// SIMATIC S7-200 SMART project (STEP 7-Micro/WIN SMART), CPU SR60

SYMBOL_TABLE A_手动
手动_测试_故障蜂鸣器1     V100.0
手动_测试_故障蜂鸣器2     V100.1
手动_测试_故障蜂鸣器3     V100.2
手动_测试_故障蜂鸣器4     V100.3
手动_测试_故障蜂鸣器5     V100.4
手动_测试_运行指示灯1     V100.5
手动_测试_运行指示灯2     V100.6
手动_测试_运行指示灯3     V100.7
手动_测试_运行指示灯4     V101.0
手动_测试_运行指示灯5     V101.1
手动_测试_停机指示灯1     V101.2
手动_测试_停机指示灯2     V101.3
手动_测试_停机指示灯3     V101.4
手动_测试_停机指示灯4     V101.5
手动_测试_停机指示灯5     V101.6
手动_测试_清洗吹扫指示1    V101.7
手动_测试_清洗吹扫指示2    V102.0
手动_测试_清洗吹扫指示3    V102.1
手动_测试_清洗吹扫指示4    V102.2
手动_测试_清洗吹扫指示5    V102.3
手动_测试_螺杆启停1      V102.4
手动_测试_螺杆启停2      V102.5
手动_测试_螺杆启停3      V102.6
手动_测试_螺杆启停4      V102.7
手动_测试_螺杆启停5      V103.0
手动_测试_入口阀1       V103.1
手动_测试_入口阀2       V103.2
手动_测试_入口阀3       V103.3
手动_测试_入口阀4       V103.4
手动_测试_入口阀5       V103.5
手动_测试_清洗阀1       V103.6
手动_测试_清洗阀2       V103.7
手动_测试_清洗阀3       V104.0
手动_测试_清洗阀4       V104.1
手动_测试_清洗阀5       V104.2
手动_测试_吹扫阀1       V104.3
手动_测试_吹扫阀2       V104.4
手动_测试_吹扫阀3       V104.5
手动_测试_吹扫阀4       V104.6
手动_测试_吹扫阀5       V104.7
END_SYMBOL_TABLE

SYMBOL_TABLE 系统符号
Always_On        SM0.0    // 始终接通
END_SYMBOL_TABLE

SYMBOL_TABLE A_自动
启动标志位1           V120.0
启动标志位2           V120.1
启动标志位3           V120.2
启动标志位4           V120.3
启动标志位5           V120.4
停机标志位1           V120.5
停机标志位2           V120.6
停机标志位3           V120.7
停机标志位4           V121.0
停机标志位5           V121.1
复位标志位1           V121.2
复位标志位2           V121.3
复位标志位3           V121.4
复位标志位4           V121.5
复位标志位5           V121.6
急停标志位1           V121.7
急停标志位2           V122.0
急停标志位3           V122.1
急停标志位4           V122.2
急停标志位5           V122.3
故障标志位1           V122.4
故障标志位2           V122.5
故障标志位3           V122.6
故障标志位4           V122.7
故障标志位5           V123.0
异常标志位1           V123.1
异常标志位2           V123.2
异常标志位3           V123.3
异常标志位4           V123.4
异常标志位5           V123.5
步骤延时触发1          V123.6
步骤延时触发2          V123.7
步骤延时触发3          V124.0
步骤延时触发4          V124.1
步骤延时触发5          V124.2
步骤延时定时器1         T37
步骤延时定时器2         T38
步骤延时定时器3         T39
步骤延时定时器4         T40
步骤延时定时器5         T41
启动前吹扫定时器1        T42
启动前吹扫定时器2        T43
启动前吹扫定时器3        T44
启动前吹扫定时器4        T45
启动前吹扫定时器5        T46
停机清洗定时器1         T47
停机清洗定时器2         T48
停机清洗定时器3         T49
停机清洗定时器4         T50
停机清洗定时器5         T51
停机吹扫定时器1         T52
停机吹扫定时器2         T53
停机吹扫定时器3         T54
停机吹扫定时器4         T55
停机吹扫定时器5         T56
自动步骤1            VW250
自动步骤2            VW252
自动步骤3            VW254
自动步骤4            VW256
自动步骤5            VW258
启动前吹扫时间_变量1      VW260
启动前吹扫时间_变量2      VW262
启动前吹扫时间_变量3      VW264
启动前吹扫时间_变量4      VW266
启动前吹扫时间_变量5      VW268
启动前吹扫时间_变量6      VW270
启动前吹扫时间_变量7      VW272
启动前吹扫时间_变量8      VW274
启动前吹扫时间_变量9      VW276
启动前吹扫时间_变量10     VW278
停机清洗时间_变量1       VW280
停机清洗时间_变量2       VW282
停机清洗时间_变量3       VW284
停机清洗时间_变量4       VW286
停机清洗时间_变量5       VW288
停机清洗时间_变量6       VW290
停机清洗时间_变量7       VW292
停机清洗时间_变量8       VW294
停机清洗时间_变量9       VW296
停机清洗时间_变量10      VW298
停机吹扫时间_变量1       VW300
停机吹扫时间_变量2       VW302
停机吹扫时间_变量3       VW304
停机吹扫时间_变量4       VW306
停机吹扫时间_变量5       VW308
停机吹扫时间_变量6       VW310
停机吹扫时间_变量7       VW312
停机吹扫时间_变量8       VW314
停机吹扫时间_变量9       VW316
停机吹扫时间_变量10      VW318
END_SYMBOL_TABLE

SYMBOL_TABLE A_参数显示_VW
启动前吹扫时间_显示1      VW500
启动前吹扫时间_显示2      VW502
启动前吹扫时间_显示3      VW504
启动前吹扫时间_显示4      VW506
启动前吹扫时间_显示5      VW508
停机清洗时间_显示1       VW510
停机清洗时间_显示2       VW512
停机清洗时间_显示3       VW514
停机清洗时间_显示4       VW516
停机清洗时间_显示5       VW518
停机吹扫时间_显示1       VW520
停机吹扫时间_显示2       VW522
停机吹扫时间_显示3       VW524
停机吹扫时间_显示4       VW526
停机吹扫时间_显示5       VW528
END_SYMBOL_TABLE

SYMBOL_TABLE A_参数设置_VD
目标真空1            VD900
目标真空2            VD904
目标真空3            VD908
目标真空4            VD912
目标真空5            VD916
入口压变上限1          VD920
入口温变上限1          VD924
冷却温变上限1          VD928
磁翻板液位上限1         VD932
入口压变上限2          VD936
入口温变上限2          VD940
冷却温变上限2          VD944
磁翻板液位上限2         VD948
入口压变上限3          VD952
入口温变上限3          VD956
冷却温变上限3          VD960
磁翻板液位上限3         VD964
入口压变上限4          VD968
入口温变上限4          VD972
冷却温变上限4          VD976
磁翻板液位上限4         VD980
入口压变上限5          VD984
入口温变上限5          VD988
冷却温变上限5          VD992
磁翻板液位上限5         VD996
END_SYMBOL_TABLE

SYMBOL_TABLE A_参数设置_VW
启动前吹扫时间_设置1      VW400
启动前吹扫时间_设置2      VW402
启动前吹扫时间_设置3      VW404
启动前吹扫时间_设置4      VW406
启动前吹扫时间_设置5      VW408
停机清洗时间_设置1       VW410
停机清洗时间_设置2       VW412
停机清洗时间_设置3       VW414
停机清洗时间_设置4       VW416
停机清洗时间_设置5       VW418
停机吹扫时间_设定1       VW420
停机吹扫时间_设定2       VW422
停机吹扫时间_设定3       VW424
停机吹扫时间_设定4       VW426
停机吹扫时间_设定5       VW428
END_SYMBOL_TABLE

SYMBOL_TABLE A_参数显示_VD
入口压力值1           VD600
入口温度值1           VD604
冷却温度值1           VD608
磁翻板液位值1          VD612
入口压力值2           VD616
入口温度值2           VD620
冷却温度值2           VD624
磁翻板液位值2          VD628
入口压力值3           VD632
入口温度值3           VD636
冷却温度值3           VD640
磁翻板液位值3          VD644
入口压力值4           VD648
入口温度值4           VD652
冷却温度值4           VD656
磁翻板液位值4          VD660
入口压力值5           VD664
入口温度值5           VD668
冷却温度值5           VD672
磁翻板液位值5          VD676
END_SYMBOL_TABLE

SUBROUTINE_BLOCK A_手动:SBR1
TITLE=子程序注释
BEGIN
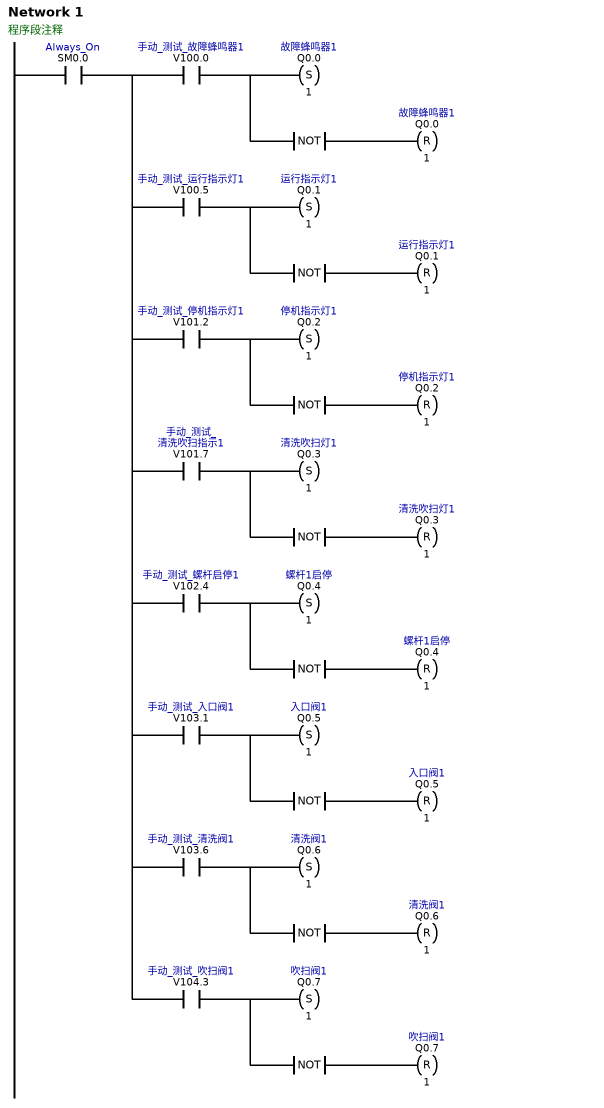
Network 1
// 程序段注释
LD     Always_On:SM0.0
LPS
A      手动_测试_故障蜂鸣器1:V100.0
S      故障蜂鸣器1:Q0.0, 1
NOT
R      故障蜂鸣器1:Q0.0, 1
LRD
A      手动_测试_运行指示灯1:V100.5
S      运行指示灯1:Q0.1, 1
NOT
R      运行指示灯1:Q0.1, 1
LRD
A      手动_测试_停机指示灯1:V101.2
S      停机指示灯1:Q0.2, 1
NOT
R      停机指示灯1:Q0.2, 1
LRD
A      手动_测试_清洗吹扫指示1:V101.7
S      清洗吹扫灯1:Q0.3, 1
NOT
R      清洗吹扫灯1:Q0.3, 1
LRD
A      手动_测试_螺杆启停1:V102.4
S      螺杆1启停:Q0.4, 1
NOT
R      螺杆1启停:Q0.4, 1
LRD
A      手动_测试_入口阀1:V103.1
S      入口阀1:Q0.5, 1
NOT
R      入口阀1:Q0.5, 1
LRD
A      手动_测试_清洗阀1:V103.6
S      清洗阀1:Q0.6, 1
NOT
R      清洗阀1:Q0.6, 1
LPP
A      手动_测试_吹扫阀1:V104.3
S      吹扫阀1:Q0.7, 1
NOT
R      吹扫阀1:Q0.7, 1
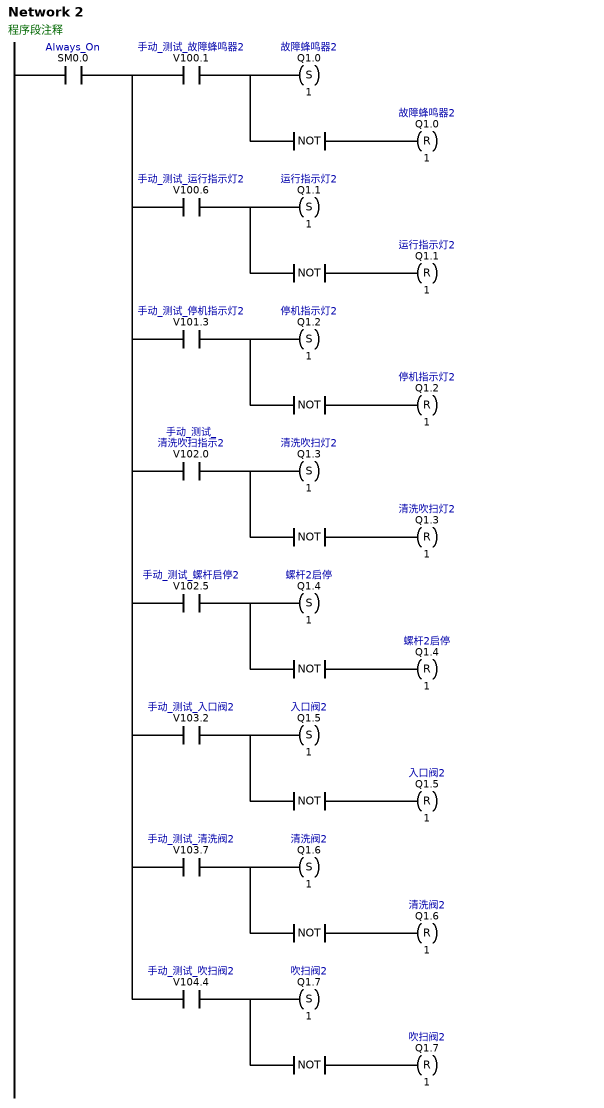
Network 2
// 程序段注释
LD     Always_On:SM0.0
LPS
A      手动_测试_故障蜂鸣器2:V100.1
S      故障蜂鸣器2:Q1.0, 1
NOT
R      故障蜂鸣器2:Q1.0, 1
LRD
A      手动_测试_运行指示灯2:V100.6
S      运行指示灯2:Q1.1, 1
NOT
R      运行指示灯2:Q1.1, 1
LRD
A      手动_测试_停机指示灯2:V101.3
S      停机指示灯2:Q1.2, 1
NOT
R      停机指示灯2:Q1.2, 1
LRD
A      手动_测试_清洗吹扫指示2:V102.0
S      清洗吹扫灯2:Q1.3, 1
NOT
R      清洗吹扫灯2:Q1.3, 1
LRD
A      手动_测试_螺杆启停2:V102.5
S      螺杆2启停:Q1.4, 1
NOT
R      螺杆2启停:Q1.4, 1
LRD
A      手动_测试_入口阀2:V103.2
S      入口阀2:Q1.5, 1
NOT
R      入口阀2:Q1.5, 1
LRD
A      手动_测试_清洗阀2:V103.7
S      清洗阀2:Q1.6, 1
NOT
R      清洗阀2:Q1.6, 1
LPP
A      手动_测试_吹扫阀2:V104.4
S      吹扫阀2:Q1.7, 1
NOT
R      吹扫阀2:Q1.7, 1
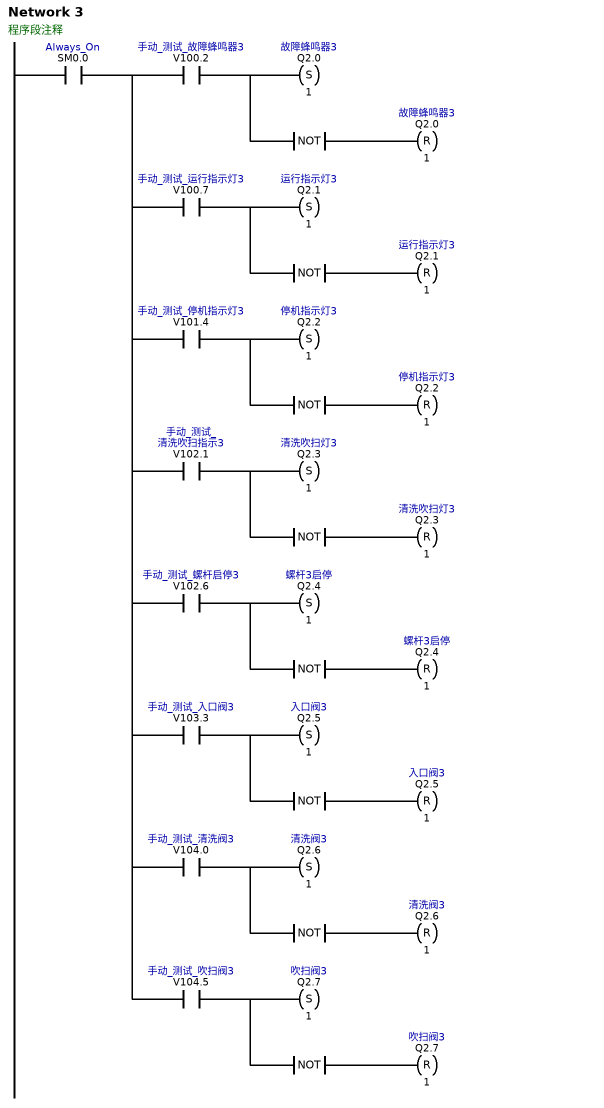
Network 3
// 程序段注释
LD     Always_On:SM0.0
LPS
A      手动_测试_故障蜂鸣器3:V100.2
S      故障蜂鸣器3:Q2.0, 1
NOT
R      故障蜂鸣器3:Q2.0, 1
LRD
A      手动_测试_运行指示灯3:V100.7
S      运行指示灯3:Q2.1, 1
NOT
R      运行指示灯3:Q2.1, 1
LRD
A      手动_测试_停机指示灯3:V101.4
S      停机指示灯3:Q2.2, 1
NOT
R      停机指示灯3:Q2.2, 1
LRD
A      手动_测试_清洗吹扫指示3:V102.1
S      清洗吹扫灯3:Q2.3, 1
NOT
R      清洗吹扫灯3:Q2.3, 1
LRD
A      手动_测试_螺杆启停3:V102.6
S      螺杆3启停:Q2.4, 1
NOT
R      螺杆3启停:Q2.4, 1
LRD
A      手动_测试_入口阀3:V103.3
S      入口阀3:Q2.5, 1
NOT
R      入口阀3:Q2.5, 1
LRD
A      手动_测试_清洗阀3:V104.0
S      清洗阀3:Q2.6, 1
NOT
R      清洗阀3:Q2.6, 1
LPP
A      手动_测试_吹扫阀3:V104.5
S      吹扫阀3:Q2.7, 1
NOT
R      吹扫阀3:Q2.7, 1
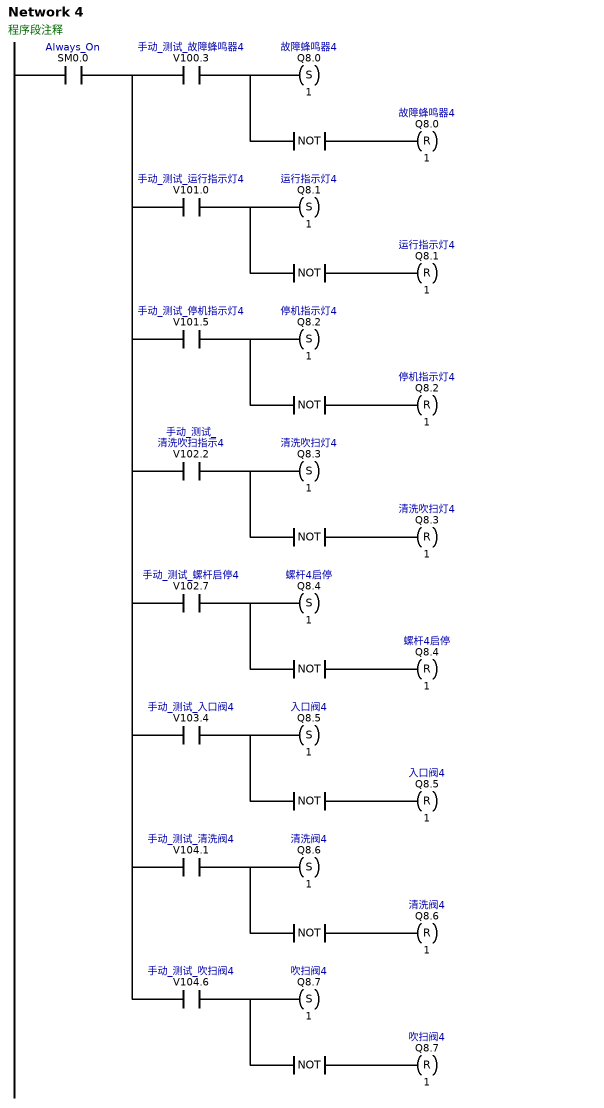
Network 4
// 程序段注释
LD     Always_On:SM0.0
LPS
A      手动_测试_故障蜂鸣器4:V100.3
S      故障蜂鸣器4:Q8.0, 1
NOT
R      故障蜂鸣器4:Q8.0, 1
LRD
A      手动_测试_运行指示灯4:V101.0
S      运行指示灯4:Q8.1, 1
NOT
R      运行指示灯4:Q8.1, 1
LRD
A      手动_测试_停机指示灯4:V101.5
S      停机指示灯4:Q8.2, 1
NOT
R      停机指示灯4:Q8.2, 1
LRD
A      手动_测试_清洗吹扫指示4:V102.2
S      清洗吹扫灯4:Q8.3, 1
NOT
R      清洗吹扫灯4:Q8.3, 1
LRD
A      手动_测试_螺杆启停4:V102.7
S      螺杆4启停:Q8.4, 1
NOT
R      螺杆4启停:Q8.4, 1
LRD
A      手动_测试_入口阀4:V103.4
S      入口阀4:Q8.5, 1
NOT
R      入口阀4:Q8.5, 1
LRD
A      手动_测试_清洗阀4:V104.1
S      清洗阀4:Q8.6, 1
NOT
R      清洗阀4:Q8.6, 1
LPP
A      手动_测试_吹扫阀4:V104.6
S      吹扫阀4:Q8.7, 1
NOT
R      吹扫阀4:Q8.7, 1
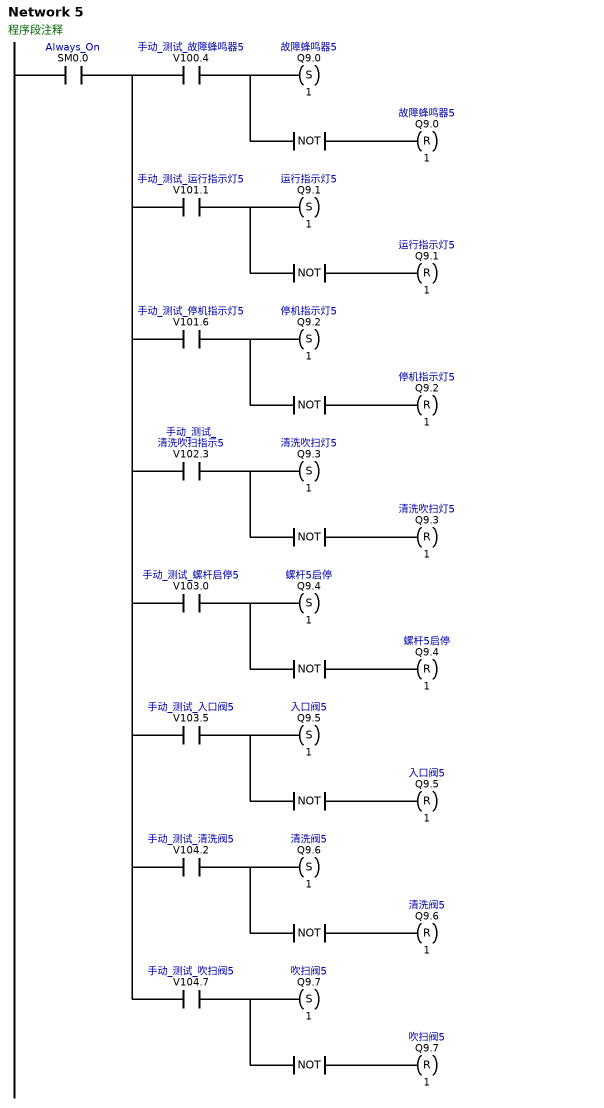
Network 5
// 程序段注释
LD     Always_On:SM0.0
LPS
A      手动_测试_故障蜂鸣器5:V100.4
S      故障蜂鸣器5:Q9.0, 1
NOT
R      故障蜂鸣器5:Q9.0, 1
LRD
A      手动_测试_运行指示灯5:V101.1
S      运行指示灯5:Q9.1, 1
NOT
R      运行指示灯5:Q9.1, 1
LRD
A      手动_测试_停机指示灯5:V101.6
S      停机指示灯5:Q9.2, 1
NOT
R      停机指示灯5:Q9.2, 1
LRD
A      手动_测试_清洗吹扫指示5:V102.3
S      清洗吹扫灯5:Q9.3, 1
NOT
R      清洗吹扫灯5:Q9.3, 1
LRD
A      手动_测试_螺杆启停5:V103.0
S      螺杆5启停:Q9.4, 1
NOT
R      螺杆5启停:Q9.4, 1
LRD
A      手动_测试_入口阀5:V103.5
S      入口阀5:Q9.5, 1
NOT
R      入口阀5:Q9.5, 1
LRD
A      手动_测试_清洗阀5:V104.2
S      清洗阀5:Q9.6, 1
NOT
R      清洗阀5:Q9.6, 1
LPP
A      手动_测试_吹扫阀5:V104.7
S      吹扫阀5:Q9.7, 1
NOT
R      吹扫阀5:Q9.7, 1
END_SUBROUTINE_BLOCK

SUBROUTINE_BLOCK A_自动:SBR2
TITLE=子程序注释
BEGIN
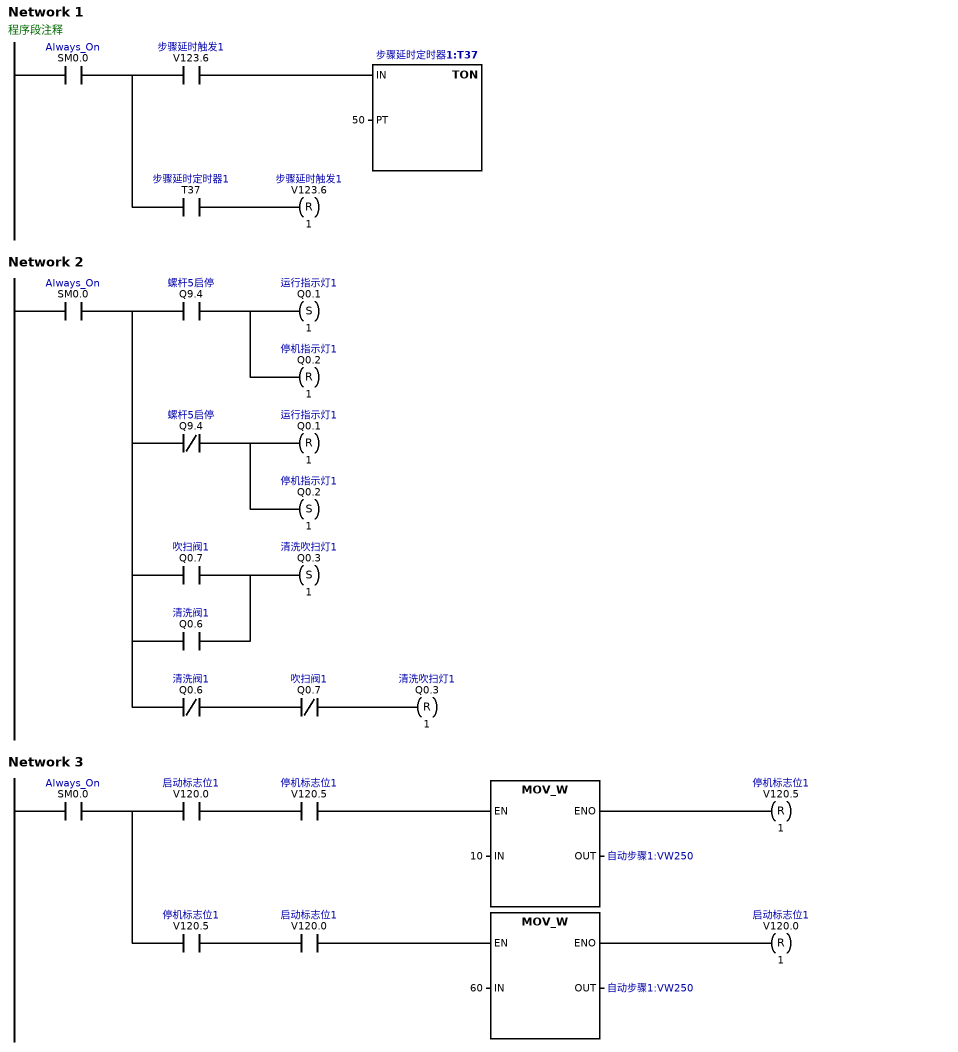
Network 1
// 程序段注释
LD     Always_On:SM0.0
LPS
A      步骤延时触发1:V123.6
TON    步骤延时定时器1:T37, 50
LPP
A      步骤延时定时器1:T37
R      步骤延时触发1:V123.6, 1
Network 2
LD     Always_On:SM0.0
LPS
A      螺杆5启停:Q9.4
S      运行指示灯1:Q0.1, 1
R      停机指示灯1:Q0.2, 1
LRD
AN     螺杆5启停:Q9.4
R      运行指示灯1:Q0.1, 1
S      停机指示灯1:Q0.2, 1
LRD
LD     吹扫阀1:Q0.7
O      清洗阀1:Q0.6
ALD
S      清洗吹扫灯1:Q0.3, 1
LPP
AN     清洗阀1:Q0.6
AN     吹扫阀1:Q0.7
R      清洗吹扫灯1:Q0.3, 1
Network 3
LD     Always_On:SM0.0
LPS
A      启动标志位1:V120.0
A      停机标志位1:V120.5
MOVW   10, 自动步骤1:VW250
AENO
R      停机标志位1:V120.5, 1
LPP
A      停机标志位1:V120.5
A      启动标志位1:V120.0
MOVW   60, 自动步骤1:VW250
AENO
R      启动标志位1:V120.0, 1
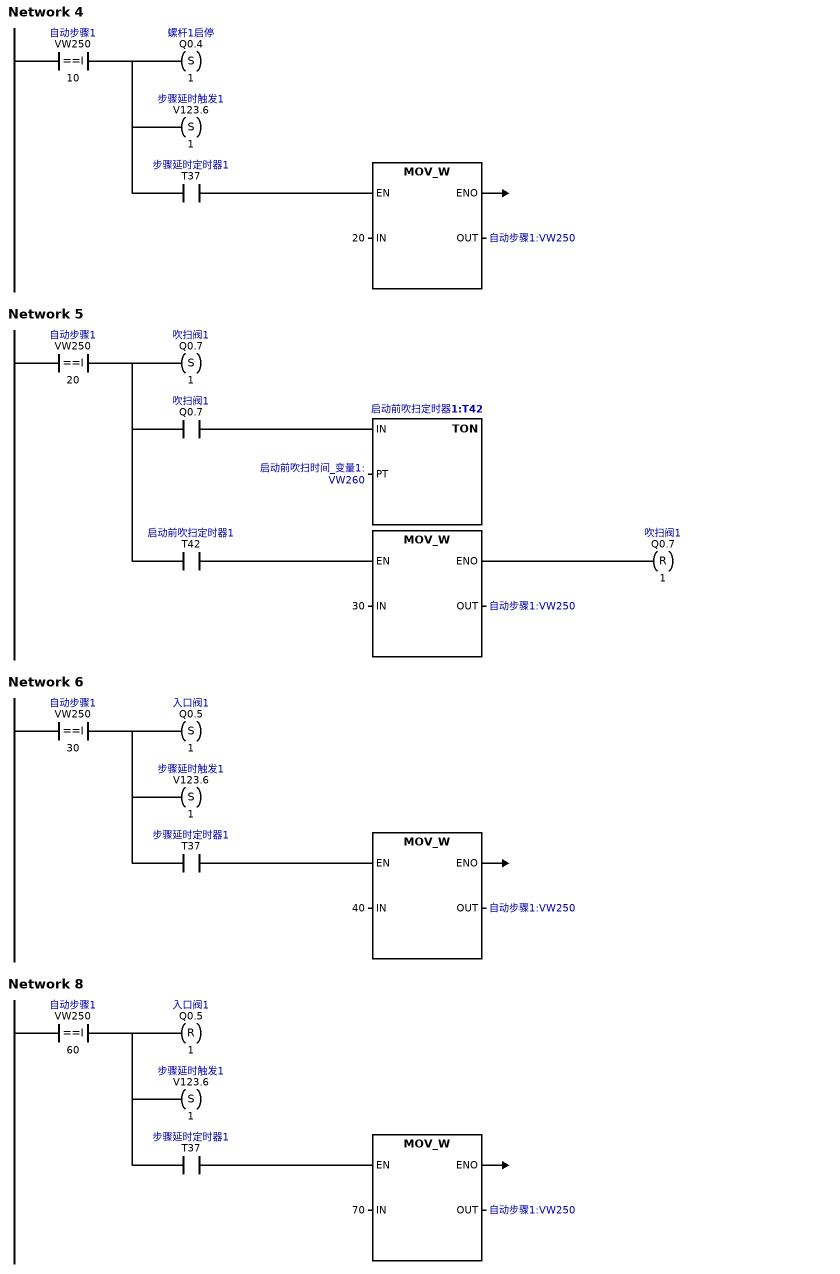
Network 4
LDW=   自动步骤1:VW250, 10
S      螺杆1启停:Q0.4, 1
S      步骤延时触发1:V123.6, 1
A      步骤延时定时器1:T37
MOVW   20, 自动步骤1:VW250
Network 5
LDW=   自动步骤1:VW250, 20
LPS
S      吹扫阀1:Q0.7, 1
A      吹扫阀1:Q0.7
TON    启动前吹扫定时器1:T42, 启动前吹扫时间_变量1:VW260
LPP
A      启动前吹扫定时器1:T42
MOVW   30, 自动步骤1:VW250
AENO
R      吹扫阀1:Q0.7, 1
Network 6
LDW=   自动步骤1:VW250, 30
S      入口阀1:Q0.5, 1
S      步骤延时触发1:V123.6, 1
A      步骤延时定时器1:T37
MOVW   40, 自动步骤1:VW250
Network 8
LDW=   自动步骤1:VW250, 60
R      入口阀1:Q0.5, 1
S      步骤延时触发1:V123.6, 1
A      步骤延时定时器1:T37
MOVW   70, 自动步骤1:VW250
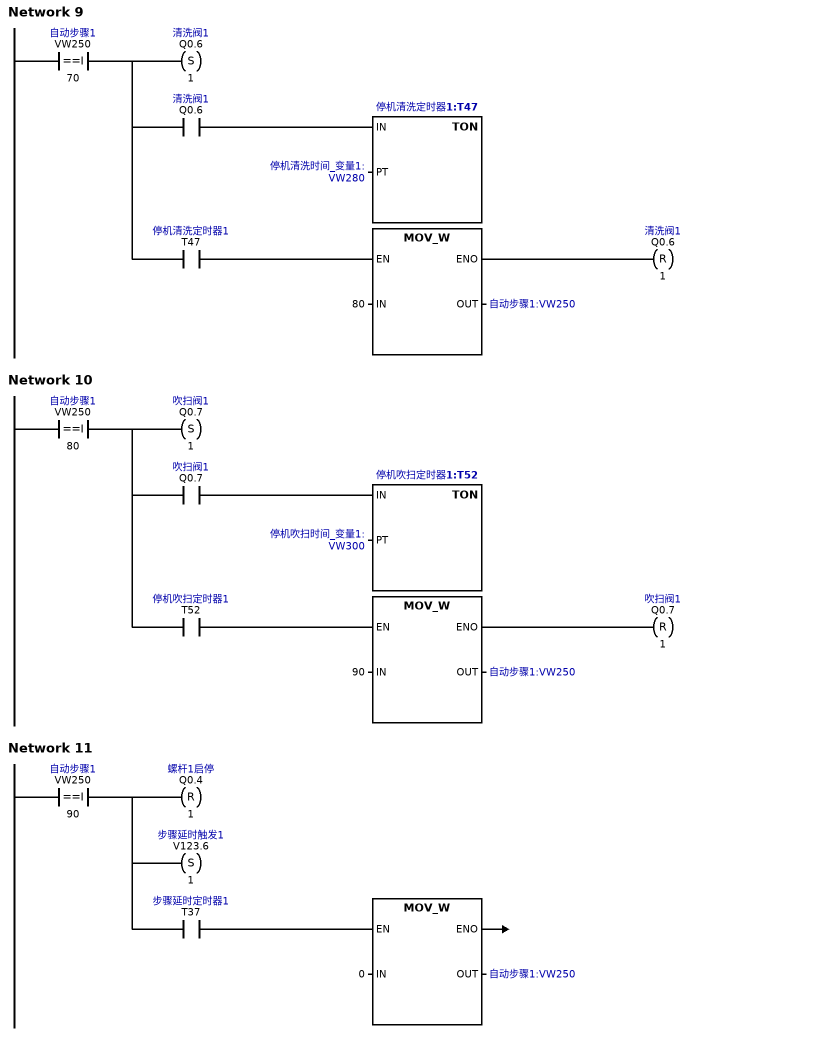
Network 9
LDW=   自动步骤1:VW250, 70
LPS
S      清洗阀1:Q0.6, 1
A      清洗阀1:Q0.6
TON    停机清洗定时器1:T47, 停机清洗时间_变量1:VW280
LPP
A      停机清洗定时器1:T47
MOVW   80, 自动步骤1:VW250
AENO
R      清洗阀1:Q0.6, 1
Network 10
LDW=   自动步骤1:VW250, 80
LPS
S      吹扫阀1:Q0.7, 1
A      吹扫阀1:Q0.7
TON    停机吹扫定时器1:T52, 停机吹扫时间_变量1:VW300
LPP
A      停机吹扫定时器1:T52
MOVW   90, 自动步骤1:VW250
AENO
R      吹扫阀1:Q0.7, 1
Network 11
LDW=   自动步骤1:VW250, 90
R      螺杆1启停:Q0.4, 1
S      步骤延时触发1:V123.6, 1
A      步骤延时定时器1:T37
MOVW   0, 自动步骤1:VW250
END_SUBROUTINE_BLOCK

SUBROUTINE_BLOCK B_定时器:SBR3
TITLE=子程序注释
BEGIN
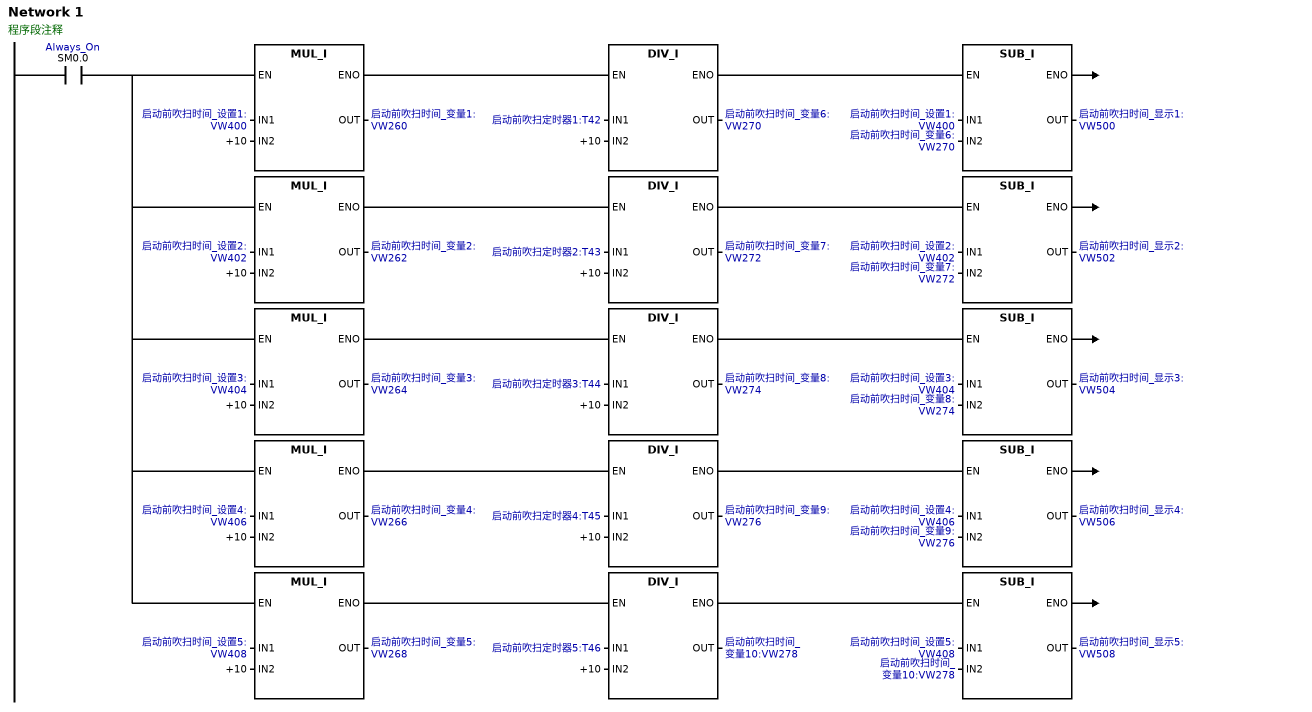
Network 1
// 程序段注释
LD     Always_On:SM0.0
LPS
MOVW   启动前吹扫时间_设置1:VW400, 启动前吹扫时间_变量1:VW260
AENO
*I     +10, 启动前吹扫时间_变量1:VW260
AENO
MOVW   启动前吹扫定时器1:T42, 启动前吹扫时间_变量6:VW270
AENO
/I     +10, 启动前吹扫时间_变量6:VW270
AENO
MOVW   启动前吹扫时间_设置1:VW400, 启动前吹扫时间_显示1:VW500
-I     启动前吹扫时间_变量6:VW270, 启动前吹扫时间_显示1:VW500
LRD
MOVW   启动前吹扫时间_设置2:VW402, 启动前吹扫时间_变量2:VW262
AENO
*I     +10, 启动前吹扫时间_变量2:VW262
AENO
MOVW   启动前吹扫定时器2:T43, 启动前吹扫时间_变量7:VW272
AENO
/I     +10, 启动前吹扫时间_变量7:VW272
AENO
MOVW   启动前吹扫时间_设置2:VW402, 启动前吹扫时间_显示2:VW502
-I     启动前吹扫时间_变量7:VW272, 启动前吹扫时间_显示2:VW502
LRD
MOVW   启动前吹扫时间_设置3:VW404, 启动前吹扫时间_变量3:VW264
AENO
*I     +10, 启动前吹扫时间_变量3:VW264
AENO
MOVW   启动前吹扫定时器3:T44, 启动前吹扫时间_变量8:VW274
AENO
/I     +10, 启动前吹扫时间_变量8:VW274
AENO
MOVW   启动前吹扫时间_设置3:VW404, 启动前吹扫时间_显示3:VW504
-I     启动前吹扫时间_变量8:VW274, 启动前吹扫时间_显示3:VW504
LRD
MOVW   启动前吹扫时间_设置4:VW406, 启动前吹扫时间_变量4:VW266
AENO
*I     +10, 启动前吹扫时间_变量4:VW266
AENO
MOVW   启动前吹扫定时器4:T45, 启动前吹扫时间_变量9:VW276
AENO
/I     +10, 启动前吹扫时间_变量9:VW276
AENO
MOVW   启动前吹扫时间_设置4:VW406, 启动前吹扫时间_显示4:VW506
-I     启动前吹扫时间_变量9:VW276, 启动前吹扫时间_显示4:VW506
LPP
MOVW   启动前吹扫时间_设置5:VW408, 启动前吹扫时间_变量5:VW268
AENO
*I     +10, 启动前吹扫时间_变量5:VW268
AENO
MOVW   启动前吹扫定时器5:T46, 启动前吹扫时间_变量10:VW278
AENO
/I     +10, 启动前吹扫时间_变量10:VW278
AENO
MOVW   启动前吹扫时间_设置5:VW408, 启动前吹扫时间_显示5:VW508
-I     启动前吹扫时间_变量10:VW278, 启动前吹扫时间_显示5:VW508
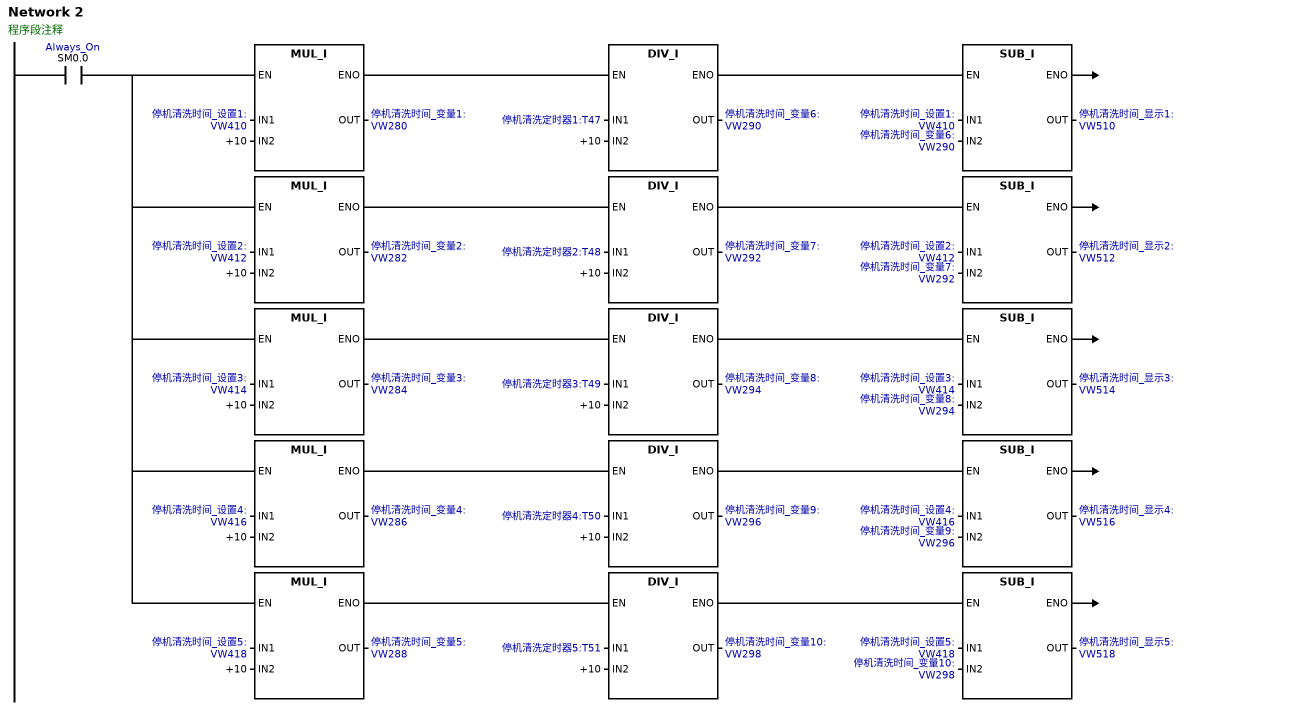
Network 2
// 程序段注释
LD     Always_On:SM0.0
LPS
MOVW   停机清洗时间_设置1:VW410, 停机清洗时间_变量1:VW280
AENO
*I     +10, 停机清洗时间_变量1:VW280
AENO
MOVW   停机清洗定时器1:T47, 停机清洗时间_变量6:VW290
AENO
/I     +10, 停机清洗时间_变量6:VW290
AENO
MOVW   停机清洗时间_设置1:VW410, 停机清洗时间_显示1:VW510
-I     停机清洗时间_变量6:VW290, 停机清洗时间_显示1:VW510
LRD
MOVW   停机清洗时间_设置2:VW412, 停机清洗时间_变量2:VW282
AENO
*I     +10, 停机清洗时间_变量2:VW282
AENO
MOVW   停机清洗定时器2:T48, 停机清洗时间_变量7:VW292
AENO
/I     +10, 停机清洗时间_变量7:VW292
AENO
MOVW   停机清洗时间_设置2:VW412, 停机清洗时间_显示2:VW512
-I     停机清洗时间_变量7:VW292, 停机清洗时间_显示2:VW512
LRD
MOVW   停机清洗时间_设置3:VW414, 停机清洗时间_变量3:VW284
AENO
*I     +10, 停机清洗时间_变量3:VW284
AENO
MOVW   停机清洗定时器3:T49, 停机清洗时间_变量8:VW294
AENO
/I     +10, 停机清洗时间_变量8:VW294
AENO
MOVW   停机清洗时间_设置3:VW414, 停机清洗时间_显示3:VW514
-I     停机清洗时间_变量8:VW294, 停机清洗时间_显示3:VW514
LRD
MOVW   停机清洗时间_设置4:VW416, 停机清洗时间_变量4:VW286
AENO
*I     +10, 停机清洗时间_变量4:VW286
AENO
MOVW   停机清洗定时器4:T50, 停机清洗时间_变量9:VW296
AENO
/I     +10, 停机清洗时间_变量9:VW296
AENO
MOVW   停机清洗时间_设置4:VW416, 停机清洗时间_显示4:VW516
-I     停机清洗时间_变量9:VW296, 停机清洗时间_显示4:VW516
LPP
MOVW   停机清洗时间_设置5:VW418, 停机清洗时间_变量5:VW288
AENO
*I     +10, 停机清洗时间_变量5:VW288
AENO
MOVW   停机清洗定时器5:T51, 停机清洗时间_变量10:VW298
AENO
/I     +10, 停机清洗时间_变量10:VW298
AENO
MOVW   停机清洗时间_设置5:VW418, 停机清洗时间_显示5:VW518
-I     停机清洗时间_变量10:VW298, 停机清洗时间_显示5:VW518
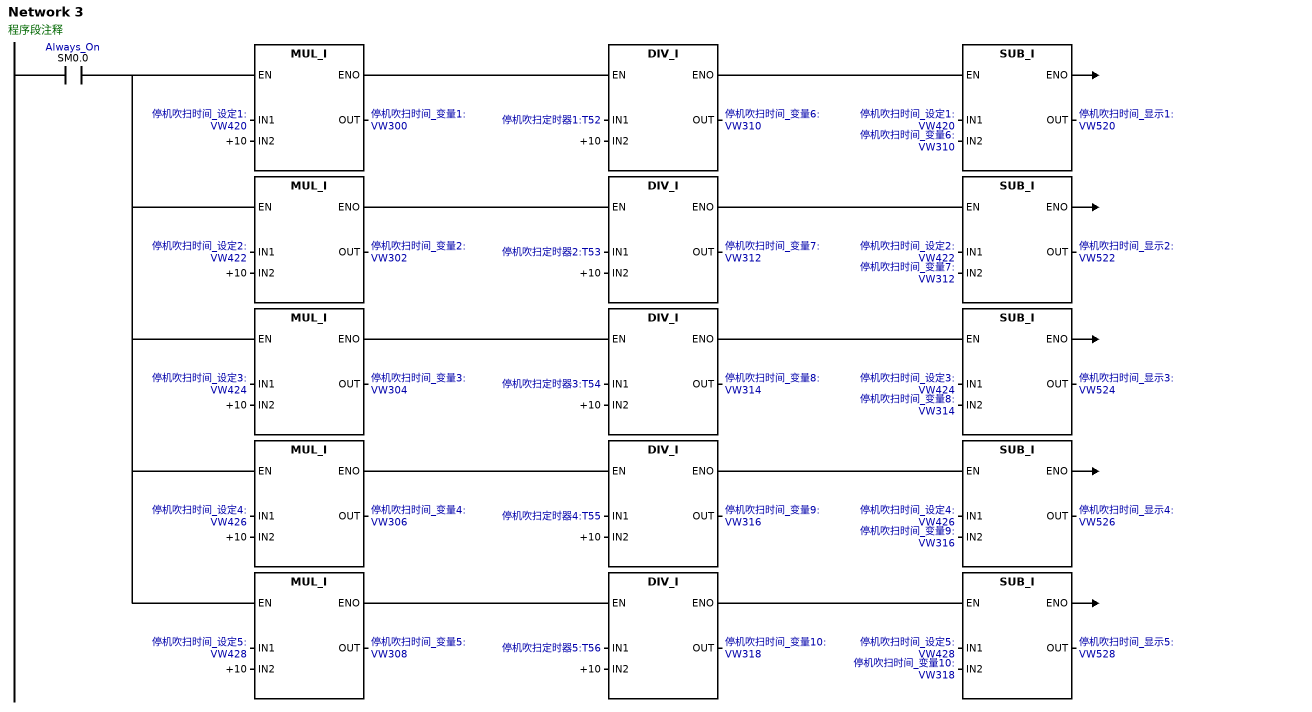
Network 3
// 程序段注释
LD     Always_On:SM0.0
LPS
MOVW   停机吹扫时间_设定1:VW420, 停机吹扫时间_变量1:VW300
AENO
*I     +10, 停机吹扫时间_变量1:VW300
AENO
MOVW   停机吹扫定时器1:T52, 停机吹扫时间_变量6:VW310
AENO
/I     +10, 停机吹扫时间_变量6:VW310
AENO
MOVW   停机吹扫时间_设定1:VW420, 停机吹扫时间_显示1:VW520
-I     停机吹扫时间_变量6:VW310, 停机吹扫时间_显示1:VW520
LRD
MOVW   停机吹扫时间_设定2:VW422, 停机吹扫时间_变量2:VW302
AENO
*I     +10, 停机吹扫时间_变量2:VW302
AENO
MOVW   停机吹扫定时器2:T53, 停机吹扫时间_变量7:VW312
AENO
/I     +10, 停机吹扫时间_变量7:VW312
AENO
MOVW   停机吹扫时间_设定2:VW422, 停机吹扫时间_显示2:VW522
-I     停机吹扫时间_变量7:VW312, 停机吹扫时间_显示2:VW522
LRD
MOVW   停机吹扫时间_设定3:VW424, 停机吹扫时间_变量3:VW304
AENO
*I     +10, 停机吹扫时间_变量3:VW304
AENO
MOVW   停机吹扫定时器3:T54, 停机吹扫时间_变量8:VW314
AENO
/I     +10, 停机吹扫时间_变量8:VW314
AENO
MOVW   停机吹扫时间_设定3:VW424, 停机吹扫时间_显示3:VW524
-I     停机吹扫时间_变量8:VW314, 停机吹扫时间_显示3:VW524
LRD
MOVW   停机吹扫时间_设定4:VW426, 停机吹扫时间_变量4:VW306
AENO
*I     +10, 停机吹扫时间_变量4:VW306
AENO
MOVW   停机吹扫定时器4:T55, 停机吹扫时间_变量9:VW316
AENO
/I     +10, 停机吹扫时间_变量9:VW316
AENO
MOVW   停机吹扫时间_设定4:VW426, 停机吹扫时间_显示4:VW526
-I     停机吹扫时间_变量9:VW316, 停机吹扫时间_显示4:VW526
LPP
MOVW   停机吹扫时间_设定5:VW428, 停机吹扫时间_变量5:VW308
AENO
*I     +10, 停机吹扫时间_变量5:VW308
AENO
MOVW   停机吹扫定时器5:T56, 停机吹扫时间_变量10:VW318
AENO
/I     +10, 停机吹扫时间_变量10:VW318
AENO
MOVW   停机吹扫时间_设定5:VW428, 停机吹扫时间_显示5:VW528
-I     停机吹扫时间_变量10:VW318, 停机吹扫时间_显示5:VW528
END_SUBROUTINE_BLOCK

// SBR4: protected block, not included

// SBR5: protected block, not included

// SBR6: protected block, not included

// SBR7: protected block, not included

// SBR8: protected block, not included

// SBR9: protected block, not included

SUBROUTINE_BLOCK A_数据采样:SBR10
TITLE=子程序注释
BEGIN
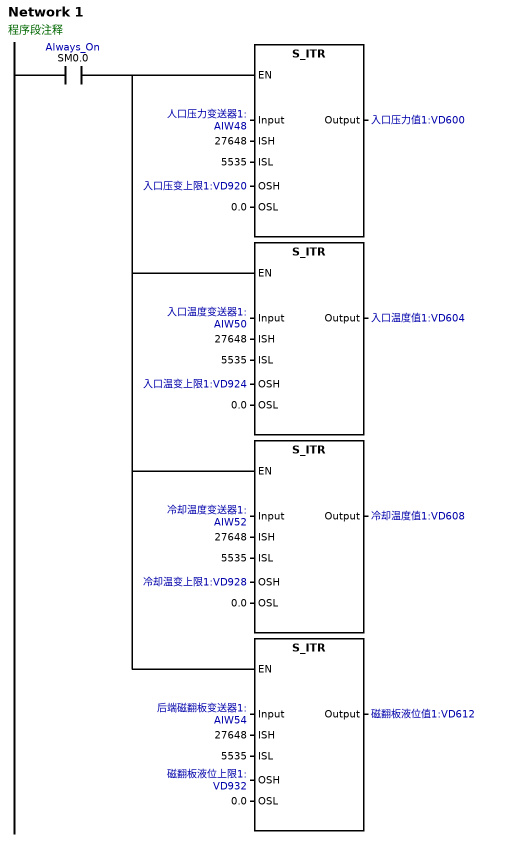
Network 1
// 程序段注释
LD     Always_On:SM0.0
CALL   S_ITR:SBR11, 人口压力变送器1:AIW48, 27648, 5535, 入口压变上限1:VD920, 0.0, 入口压力值1:VD600
CALL   S_ITR:SBR11, 入口温度变送器1:AIW50, 27648, 5535, 入口温变上限1:VD924, 0.0, 入口温度值1:VD604
CALL   S_ITR:SBR11, 冷却温度变送器1:AIW52, 27648, 5535, 冷却温变上限1:VD928, 0.0, 冷却温度值1:VD608
CALL   S_ITR:SBR11, 后端磁翻板变送器1:AIW54, 27648, 5535, 磁翻板液位上限1:VD932, 0.0, 磁翻板液位值1:VD612
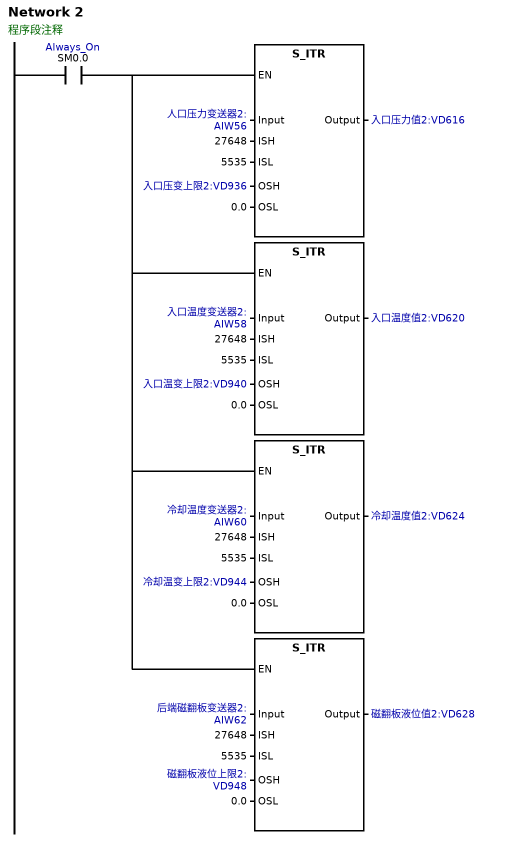
Network 2
// 程序段注释
LD     Always_On:SM0.0
CALL   S_ITR:SBR11, 人口压力变送器2:AIW56, 27648, 5535, 入口压变上限2:VD936, 0.0, 入口压力值2:VD616
CALL   S_ITR:SBR11, 入口温度变送器2:AIW58, 27648, 5535, 入口温变上限2:VD940, 0.0, 入口温度值2:VD620
CALL   S_ITR:SBR11, 冷却温度变送器2:AIW60, 27648, 5535, 冷却温变上限2:VD944, 0.0, 冷却温度值2:VD624
CALL   S_ITR:SBR11, 后端磁翻板变送器2:AIW62, 27648, 5535, 磁翻板液位上限2:VD948, 0.0, 磁翻板液位值2:VD628
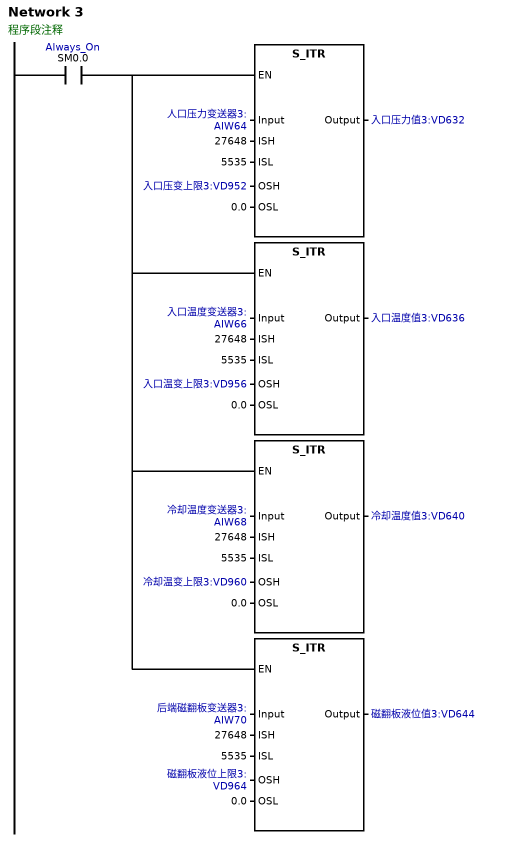
Network 3
// 程序段注释
LD     Always_On:SM0.0
CALL   S_ITR:SBR11, 人口压力变送器3:AIW64, 27648, 5535, 入口压变上限3:VD952, 0.0, 入口压力值3:VD632
CALL   S_ITR:SBR11, 入口温度变送器3:AIW66, 27648, 5535, 入口温变上限3:VD956, 0.0, 入口温度值3:VD636
CALL   S_ITR:SBR11, 冷却温度变送器3:AIW68, 27648, 5535, 冷却温变上限3:VD960, 0.0, 冷却温度值3:VD640
CALL   S_ITR:SBR11, 后端磁翻板变送器3:AIW70, 27648, 5535, 磁翻板液位上限3:VD964, 0.0, 磁翻板液位值3:VD644
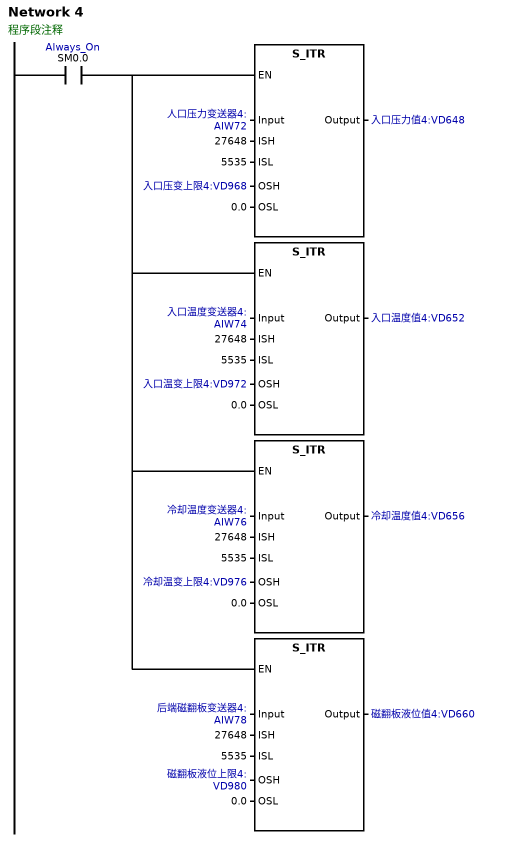
Network 4
// 程序段注释
LD     Always_On:SM0.0
CALL   S_ITR:SBR11, 人口压力变送器4:AIW72, 27648, 5535, 入口压变上限4:VD968, 0.0, 入口压力值4:VD648
CALL   S_ITR:SBR11, 入口温度变送器4:AIW74, 27648, 5535, 入口温变上限4:VD972, 0.0, 入口温度值4:VD652
CALL   S_ITR:SBR11, 冷却温度变送器4:AIW76, 27648, 5535, 冷却温变上限4:VD976, 0.0, 冷却温度值4:VD656
CALL   S_ITR:SBR11, 后端磁翻板变送器4:AIW78, 27648, 5535, 磁翻板液位上限4:VD980, 0.0, 磁翻板液位值4:VD660
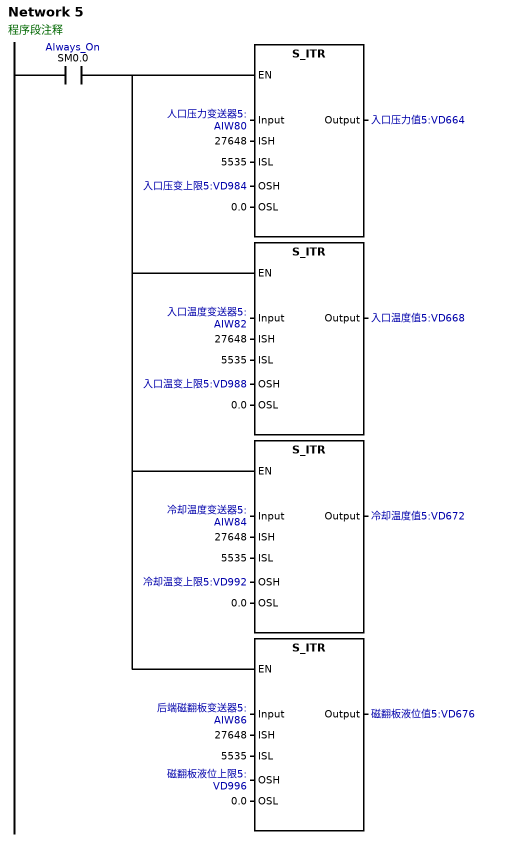
Network 5
// 程序段注释
LD     Always_On:SM0.0
CALL   S_ITR:SBR11, 人口压力变送器5:AIW80, 27648, 5535, 入口压变上限5:VD984, 0.0, 入口压力值5:VD664
CALL   S_ITR:SBR11, 入口温度变送器5:AIW82, 27648, 5535, 入口温变上限5:VD988, 0.0, 入口温度值5:VD668
CALL   S_ITR:SBR11, 冷却温度变送器5:AIW84, 27648, 5535, 冷却温变上限5:VD992, 0.0, 冷却温度值5:VD672
CALL   S_ITR:SBR11, 后端磁翻板变送器5:AIW86, 27648, 5535, 磁翻板液位上限5:VD996, 0.0, 磁翻板液位值5:VD676
END_SUBROUTINE_BLOCK

// SBR11: protected block, not included

// INT1: protected block, not included
